(* IEC 61131-3 sources: SafePLC-Gen-Evaluation/Evaluation Results/eastman/run_05, 2 files *)

(* ---- io_declarations.st ---- *)
(* ==================================================  *)
(* PLC I/O Variable Declarations — CODESYS 3.5  *)
(* Generated by SafePLC-Gen Multimodal  *)
(* ==================================================  *)

VAR_GLOBAL
    (* --- Analog Inputs ---  *)
    FI_1_Raw                     AT %IW0       : INT := 0;    (* FI-1 — Flow indicator on feed/process line P-65  *)
    FI_2_Raw                     AT %IW2       : INT := 0;    (* FI-2 — Flow indicator on line P-54/P-52 area, f  *)
    FI_3_Raw                     AT %IW4       : INT := 0;    (* FI-3 — Flow indicator on line P-57 area, Column  *)
    TI_1_Raw                     AT %IW6       : INT := 0;    (* TI-1 — Temperature indicator, bottom-left area   *)
    TI_4_Raw                     AT %IW8       : INT := 0;    (* TI-4 — Temperature indicator on feed line to Co  *)
    TI_5_Raw                     AT %IW10      : INT := 0;    (* TI-5 — Temperature indicator on Column 2 (E-7),  *)
    TI_6_Raw                     AT %IW12      : INT := 0;    (* TI-6 — Temperature indicator on separator E-18   *)
    TI_7_Raw                     AT %IW14      : INT := 0;    (* TI-7 — Temperature indicator on Column 3 or ves  *)
    TI_8_Raw                     AT %IW16      : INT := 0;    (* TI-8 — Temperature indicator on Column 3, upper  *)
    (* --- Analog Outputs ---  *)
    V_3_Out                      AT %QW0       : INT := 0;    (* V-3 — Control valve on line P-28/P-73 from dec  *)
    V_4_Out                      AT %QW2       : INT := 0;    (* V-4 — Control valve on line P-74/P-12 feed to   *)
    V_5_Out                      AT %QW4       : INT := 0;    (* V-5 — Control valve on overhead/reflux line P-  *)
    V_7_Out                      AT %QW6       : INT := 0;    (* V-7 — Control valve on line P-19 from separato  *)
END_VAR

(* ---- generated_code.st ---- *)
(* Generated by SafePLC-Gen Multimodal — CODESYS 3.5 *)
(* IEC 61131-3 Structured Text *)
(* Date: 2026-04-25T12:43:58.560340 *)

PROGRAM DistillationControl

VAR
    FI_1_Raw                     AT %IW0       : INT := 0;
    FI_2_Raw                     AT %IW2       : INT := 0;
    FI_3_Raw                     AT %IW4       : INT := 0;
    TI_1_Raw                     AT %IW6       : INT := 0;
    TI_4_Raw                     AT %IW8       : INT := 0;
    TI_5_Raw                     AT %IW10      : INT := 0;
    TI_6_Raw                     AT %IW12      : INT := 0;
    TI_7_Raw                     AT %IW14      : INT := 0;
    TI_8_Raw                     AT %IW16      : INT := 0;
    V_3_Out                      AT %QW0       : INT := 0;
    V_4_Out                      AT %QW2       : INT := 0;
    V_5_Out                      AT %QW4       : INT := 0;
    V_7_Out                      AT %QW6       : INT := 0;
END_VAR

VAR
    FirstScan                    : BOOL := TRUE;

    FI_1_Scaled                  : REAL := 0.0;
    FI_2_Scaled                  : REAL := 0.0;
    FI_3_Scaled                  : REAL := 0.0;
    TI_1_Scaled                  : REAL := 0.0;
    TI_4_Scaled                  : REAL := 0.0;
    TI_5_Scaled                  : REAL := 0.0;
    TI_6_Scaled                  : REAL := 0.0;
    TI_7_Scaled                  : REAL := 0.0;
    TI_8_Scaled                  : REAL := 0.0;

    FI_1_HH_SP                   : REAL := 120.0;
    FI_1_H_SP                    : REAL := 100.0;
    FI_1_L_SP                    : REAL := 20.0;
    FI_1_LL_SP                   : REAL := 10.0;
    FI_1_Deadband                : REAL := 2.0;
    FI_1_HH                      : BOOL := FALSE;
    FI_1_H                       : BOOL := FALSE;
    FI_1_L                       : BOOL := FALSE;
    FI_1_LL                      : BOOL := FALSE;
    FI_1_HH_Latch                : SR := (S1 := FALSE, R := FALSE);
    FI_1_LL_Latch                : SR := (S1 := FALSE, R := FALSE);
    FI_1_HH_Ack                  : BOOL := FALSE;
    FI_1_LL_Ack                  : BOOL := FALSE;

    FI_2_HH_SP                   : REAL := 120.0;
    FI_2_H_SP                    : REAL := 100.0;
    FI_2_L_SP                    : REAL := 20.0;
    FI_2_LL_SP                   : REAL := 10.0;
    FI_2_Deadband                : REAL := 2.0;
    FI_2_HH                      : BOOL := FALSE;
    FI_2_H                       : BOOL := FALSE;
    FI_2_L                       : BOOL := FALSE;
    FI_2_LL                      : BOOL := FALSE;
    FI_2_HH_Latch                : SR := (S1 := FALSE, R := FALSE);
    FI_2_LL_Latch                : SR := (S1 := FALSE, R := FALSE);
    FI_2_HH_Ack                  : BOOL := FALSE;
    FI_2_LL_Ack                  : BOOL := FALSE;

    FI_3_HH_SP                   : REAL := 120.0;
    FI_3_H_SP                    : REAL := 100.0;
    FI_3_L_SP                    : REAL := 20.0;
    FI_3_LL_SP                   : REAL := 10.0;
    FI_3_Deadband                : REAL := 2.0;
    FI_3_HH                      : BOOL := FALSE;
    FI_3_H                       : BOOL := FALSE;
    FI_3_L                       : BOOL := FALSE;
    FI_3_LL                      : BOOL := FALSE;
    FI_3_HH_Latch                : SR := (S1 := FALSE, R := FALSE);
    FI_3_LL_Latch                : SR := (S1 := FALSE, R := FALSE);
    FI_3_HH_Ack                  : BOOL := FALSE;
    FI_3_LL_Ack                  : BOOL := FALSE;

    TI_1_HH_SP                   : REAL := 120.0;
    TI_1_H_SP                    : REAL := 110.0;
    TI_1_L_SP                    : REAL := 40.0;
    TI_1_LL_SP                   : REAL := 30.0;
    TI_1_Deadband                : REAL := 1.0;
    TI_1_HH                      : BOOL := FALSE;
    TI_1_H                       : BOOL := FALSE;
    TI_1_L                       : BOOL := FALSE;
    TI_1_LL                      : BOOL := FALSE;
    TI_1_HH_Latch                : SR := (S1 := FALSE, R := FALSE);
    TI_1_LL_Latch                : SR := (S1 := FALSE, R := FALSE);
    TI_1_HH_Ack                  : BOOL := FALSE;
    TI_1_LL_Ack                  : BOOL := FALSE;

    TI_4_HH_SP                   : REAL := 120.0;
    TI_4_H_SP                    : REAL := 110.0;
    TI_4_L_SP                    : REAL := 40.0;
    TI_4_LL_SP                   : REAL := 30.0;
    TI_4_Deadband                : REAL := 1.0;
    TI_4_HH                      : BOOL := FALSE;
    TI_4_H                       : BOOL := FALSE;
    TI_4_L                       : BOOL := FALSE;
    TI_4_LL                      : BOOL := FALSE;
    TI_4_HH_Latch                : SR := (S1 := FALSE, R := FALSE);
    TI_4_LL_Latch                : SR := (S1 := FALSE, R := FALSE);
    TI_4_HH_Ack                  : BOOL := FALSE;
    TI_4_LL_Ack                  : BOOL := FALSE;

    TI_5_HH_SP                   : REAL := 120.0;
    TI_5_H_SP                    : REAL := 110.0;
    TI_5_L_SP                    : REAL := 40.0;
    TI_5_LL_SP                   : REAL := 30.0;
    TI_5_Deadband                : REAL := 1.0;
    TI_5_HH                      : BOOL := FALSE;
    TI_5_H                       : BOOL := FALSE;
    TI_5_L                       : BOOL := FALSE;
    TI_5_LL                      : BOOL := FALSE;
    TI_5_HH_Latch                : SR := (S1 := FALSE, R := FALSE);
    TI_5_LL_Latch                : SR := (S1 := FALSE, R := FALSE);
    TI_5_HH_Ack                  : BOOL := FALSE;
    TI_5_LL_Ack                  : BOOL := FALSE;

    TI_6_HH_SP                   : REAL := 120.0;
    TI_6_H_SP                    : REAL := 110.0;
    TI_6_L_SP                    : REAL := 40.0;
    TI_6_LL_SP                   : REAL := 30.0;
    TI_6_Deadband                : REAL := 1.0;
    TI_6_HH                      : BOOL := FALSE;
    TI_6_H                       : BOOL := FALSE;
    TI_6_L                       : BOOL := FALSE;
    TI_6_LL                      : BOOL := FALSE;
    TI_6_HH_Latch                : SR := (S1 := FALSE, R := FALSE);
    TI_6_LL_Latch                : SR := (S1 := FALSE, R := FALSE);
    TI_6_HH_Ack                  : BOOL := FALSE;
    TI_6_LL_Ack                  : BOOL := FALSE;

    TI_7_HH_SP                   : REAL := 120.0;
    TI_7_H_SP                    : REAL := 110.0;
    TI_7_L_SP                    : REAL := 40.0;
    TI_7_LL_SP                   : REAL := 30.0;
    TI_7_Deadband                : REAL := 1.0;
    TI_7_HH                      : BOOL := FALSE;
    TI_7_H                       : BOOL := FALSE;
    TI_7_L                       : BOOL := FALSE;
    TI_7_LL                      : BOOL := FALSE;
    TI_7_HH_Latch                : SR := (S1 := FALSE, R := FALSE);
    TI_7_LL_Latch                : SR := (S1 := FALSE, R := FALSE);
    TI_7_HH_Ack                  : BOOL := FALSE;
    TI_7_LL_Ack                  : BOOL := FALSE;

    TI_8_HH_SP                   : REAL := 120.0;
    TI_8_H_SP                    : REAL := 110.0;
    TI_8_L_SP                    : REAL := 40.0;
    TI_8_LL_SP                   : REAL := 30.0;
    TI_8_Deadband                : REAL := 1.0;
    TI_8_HH                      : BOOL := FALSE;
    TI_8_H                       : BOOL := FALSE;
    TI_8_L                       : BOOL := FALSE;
    TI_8_LL                      : BOOL := FALSE;
    TI_8_HH_Latch                : SR := (S1 := FALSE, R := FALSE);
    TI_8_LL_Latch                : SR := (S1 := FALSE, R := FALSE);
    TI_8_HH_Ack                  : BOOL := FALSE;
    TI_8_LL_Ack                  : BOOL := FALSE;

    FC1_SP                       : REAL := 50.0;
    FC1_Kp                       : REAL := 1.2;
    FC1_Ki                       : REAL := 0.05;
    FC1_Error                    : REAL := 0.0;
    FC1_Integral                 : REAL := 0.0;
    FC1_Output                   : REAL := 0.0;

    FC2_SP                       : REAL := 50.0;
    FC2_Kp                       : REAL := 1.2;
    FC2_Ki                       : REAL := 0.05;
    FC2_Error                    : REAL := 0.0;
    FC2_Integral                 : REAL := 0.0;
    FC2_Output                   : REAL := 0.0;

    FC3_SP                       : REAL := 50.0;
    FC3_Kp                       : REAL := 1.2;
    FC3_Ki                       : REAL := 0.05;
    FC3_Error                    : REAL := 0.0;
    FC3_Integral                 : REAL := 0.0;
    FC3_Output                   : REAL := 0.0;

    TC1_SP                       : REAL := 80.0;
    TC1_Kp                       : REAL := 1.0;
    TC1_Ki                       : REAL := 0.03;
    TC1_Error                    : REAL := 0.0;
    TC1_Integral                 : REAL := 0.0;
    TC1_Output                   : REAL := 0.0;

    System_Alarm                 : BOOL := FALSE;
END_VAR

IF FirstScan THEN
    V_3_Out          := 6554;
    V_4_Out          := 6554;
    V_5_Out          := 6554;
    V_7_Out          := 6554;
    FC1_Integral     := 0.0;
    FC2_Integral     := 0.0;
    FC3_Integral     := 0.0;
    TC1_Integral     := 0.0;
    FI_1_HH_Latch(S1 := FALSE, R := FALSE);
    FI_1_LL_Latch(S1 := FALSE, R := FALSE);
    FI_2_HH_Latch(S1 := FALSE, R := FALSE);
    FI_2_LL_Latch(S1 := FALSE, R := FALSE);
    FI_3_HH_Latch(S1 := FALSE, R := FALSE);
    FI_3_LL_Latch(S1 := FALSE, R := FALSE);
    TI_1_HH_Latch(S1 := FALSE, R := FALSE);
    TI_1_LL_Latch(S1 := FALSE, R := FALSE);
    TI_4_HH_Latch(S1 := FALSE, R := FALSE);
    TI_4_LL_Latch(S1 := FALSE, R := FALSE);
    TI_5_HH_Latch(S1 := FALSE, R := FALSE);
    TI_5_LL_Latch(S1 := FALSE, R := FALSE);
    TI_6_HH_Latch(S1 := FALSE, R := FALSE);
    TI_6_LL_Latch(S1 := FALSE, R := FALSE);
    TI_7_HH_Latch(S1 := FALSE, R := FALSE);
    TI_7_LL_Latch(S1 := FALSE, R := FALSE);
    TI_8_HH_Latch(S1 := FALSE, R := FALSE);
    TI_8_LL_Latch(S1 := FALSE, R := FALSE);
    FirstScan        := FALSE;
    RETURN;
END_IF;

FI_1_Scaled := ((INT_TO_REAL(FI_1_Raw) - 6554.0) / (32767.0 - 6554.0)) * 150.0;
FI_2_Scaled := ((INT_TO_REAL(FI_2_Raw) - 6554.0) / (32767.0 - 6554.0)) * 150.0;
FI_3_Scaled := ((INT_TO_REAL(FI_3_Raw) - 6554.0) / (32767.0 - 6554.0)) * 150.0;
TI_1_Scaled := ((INT_TO_REAL(TI_1_Raw) - 6554.0) / (32767.0 - 6554.0)) * 150.0;
TI_4_Scaled := ((INT_TO_REAL(TI_4_Raw) - 6554.0) / (32767.0 - 6554.0)) * 150.0;
TI_5_Scaled := ((INT_TO_REAL(TI_5_Raw) - 6554.0) / (32767.0 - 6554.0)) * 150.0;
TI_6_Scaled := ((INT_TO_REAL(TI_6_Raw) - 6554.0) / (32767.0 - 6554.0)) * 150.0;
TI_7_Scaled := ((INT_TO_REAL(TI_7_Raw) - 6554.0) / (32767.0 - 6554.0)) * 150.0;
TI_8_Scaled := ((INT_TO_REAL(TI_8_Raw) - 6554.0) / (32767.0 - 6554.0)) * 150.0;

IF FI_1_Scaled >= FI_1_HH_SP THEN
    FI_1_HH_Latch.S1 := TRUE;
ELSIF FI_1_Scaled <= (FI_1_HH_SP - FI_1_Deadband) THEN
    FI_1_HH_Latch.S1 := FALSE;
END_IF;
FI_1_HH_Latch.R := FI_1_HH_Ack AND (FI_1_Scaled < FI_1_HH_SP);
FI_1_HH_Latch(S1 := FI_1_HH_Latch.S1, R := FI_1_HH_Latch.R);
FI_1_HH := FI_1_HH_Latch.Q1;

IF FI_1_Scaled >= FI_1_H_SP THEN
    FI_1_H := TRUE;
ELSIF FI_1_Scaled < (FI_1_H_SP - FI_1_Deadband) THEN
    FI_1_H := FALSE;
END_IF;

IF FI_1_Scaled <= FI_1_LL_SP THEN
    FI_1_LL_Latch.S1 := TRUE;
ELSIF FI_1_Scaled >= (FI_1_LL_SP + FI_1_Deadband) THEN
    FI_1_LL_Latch.S1 := FALSE;
END_IF;
FI_1_LL_Latch.R := FI_1_LL_Ack AND (FI_1_Scaled > FI_1_LL_SP);
FI_1_LL_Latch(S1 := FI_1_LL_Latch.S1, R := FI_1_LL_Latch.R);
FI_1_LL := FI_1_LL_Latch.Q1;

IF FI_1_Scaled <= FI_1_L_SP THEN
    FI_1_L := TRUE;
ELSIF FI_1_Scaled > (FI_1_L_SP + FI_1_Deadband) THEN
    FI_1_L := FALSE;
END_IF;

IF FI_2_Scaled >= FI_2_HH_SP THEN
    FI_2_HH_Latch.S1 := TRUE;
ELSIF FI_2_Scaled <= (FI_2_HH_SP - FI_2_Deadband) THEN
    FI_2_HH_Latch.S1 := FALSE;
END_IF;
FI_2_HH_Latch.R := FI_2_HH_Ack AND (FI_2_Scaled < FI_2_HH_SP);
FI_2_HH_Latch(S1 := FI_2_HH_Latch.S1, R := FI_2_HH_Latch.R);
FI_2_HH := FI_2_HH_Latch.Q1;

IF FI_2_Scaled >= FI_2_H_SP THEN
    FI_2_H := TRUE;
ELSIF FI_2_Scaled < (FI_2_H_SP - FI_2_Deadband) THEN
    FI_2_H := FALSE;
END_IF;

IF FI_2_Scaled <= FI_2_LL_SP THEN
    FI_2_LL_Latch.S1 := TRUE;
ELSIF FI_2_Scaled >= (FI_2_LL_SP + FI_2_Deadband) THEN
    FI_2_LL_Latch.S1 := FALSE;
END_IF;
FI_2_LL_Latch.R := FI_2_LL_Ack AND (FI_2_Scaled > FI_2_LL_SP);
FI_2_LL_Latch(S1 := FI_2_LL_Latch.S1, R := FI_2_LL_Latch.R);
FI_2_LL := FI_2_LL_Latch.Q1;

IF FI_2_Scaled <= FI_2_L_SP THEN
    FI_2_L := TRUE;
ELSIF FI_2_Scaled > (FI_2_L_SP + FI_2_Deadband) THEN
    FI_2_L := FALSE;
END_IF;

IF FI_3_Scaled >= FI_3_HH_SP THEN
    FI_3_HH_Latch.S1 := TRUE;
ELSIF FI_3_Scaled <= (FI_3_HH_SP - FI_3_Deadband) THEN
    FI_3_HH_Latch.S1 := FALSE;
END_IF;
FI_3_HH_Latch.R := FI_3_HH_Ack AND (FI_3_Scaled < FI_3_HH_SP);
FI_3_HH_Latch(S1 := FI_3_HH_Latch.S1, R := FI_3_HH_Latch.R);
FI_3_HH := FI_3_HH_Latch.Q1;

IF FI_3_Scaled >= FI_3_H_SP THEN
    FI_3_H := TRUE;
ELSIF FI_3_Scaled < (FI_3_H_SP - FI_3_Deadband) THEN
    FI_3_H := FALSE;
END_IF;

IF FI_3_Scaled <= FI_3_LL_SP THEN
    FI_3_LL_Latch.S1 := TRUE;
ELSIF FI_3_Scaled >= (FI_3_LL_SP + FI_3_Deadband) THEN
    FI_3_LL_Latch.S1 := FALSE;
END_IF;
FI_3_LL_Latch.R := FI_3_LL_Ack AND (FI_3_Scaled > FI_3_LL_SP);
FI_3_LL_Latch(S1 := FI_3_LL_Latch.S1, R := FI_3_LL_Latch.R);
FI_3_LL := FI_3_LL_Latch.Q1;

IF FI_3_Scaled <= FI_3_L_SP THEN
    FI_3_L := TRUE;
ELSIF FI_3_Scaled > (FI_3_L_SP + FI_3_Deadband) THEN
    FI_3_L := FALSE;
END_IF;

IF TI_1_Scaled >= TI_1_HH_SP THEN
    TI_1_HH_Latch.S1 := TRUE;
ELSIF TI_1_Scaled <= (TI_1_HH_SP - TI_1_Deadband) THEN
    TI_1_HH_Latch.S1 := FALSE;
END_IF;
TI_1_HH_Latch.R := TI_1_HH_Ack AND (TI_1_Scaled < TI_1_HH_SP);
TI_1_HH_Latch(S1 := TI_1_HH_Latch.S1, R := TI_1_HH_Latch.R);
TI_1_HH := TI_1_HH_Latch.Q1;

IF TI_1_Scaled >= TI_1_H_SP THEN
    TI_1_H := TRUE;
ELSIF TI_1_Scaled < (TI_1_H_SP - TI_1_Deadband) THEN
    TI_1_H := FALSE;
END_IF;

IF TI_1_Scaled <= TI_1_LL_SP THEN
    TI_1_LL_Latch.S1 := TRUE;
ELSIF TI_1_Scaled >= (TI_1_LL_SP + TI_1_Deadband) THEN
    TI_1_LL_Latch.S1 := FALSE;
END_IF;
TI_1_LL_Latch.R := TI_1_LL_Ack AND (TI_1_Scaled > TI_1_LL_SP);
TI_1_LL_Latch(S1 := TI_1_LL_Latch.S1, R := TI_1_LL_Latch.R);
TI_1_LL := TI_1_LL_Latch.Q1;

IF TI_1_Scaled <= TI_1_L_SP THEN
    TI_1_L := TRUE;
ELSIF TI_1_Scaled > (TI_1_L_SP + TI_1_Deadband) THEN
    TI_1_L := FALSE;
END_IF;

IF TI_4_Scaled >= TI_4_HH_SP THEN
    TI_4_HH_Latch.S1 := TRUE;
ELSIF TI_4_Scaled <= (TI_4_HH_SP - TI_4_Deadband) THEN
    TI_4_HH_Latch.S1 := FALSE;
END_IF;
TI_4_HH_Latch.R := TI_4_HH_Ack AND (TI_4_Scaled < TI_4_HH_SP);
TI_4_HH_Latch(S1 := TI_4_HH_Latch.S1, R := TI_4_HH_Latch.R);
TI_4_HH := TI_4_HH_Latch.Q1;

IF TI_4_Scaled >= TI_4_H_SP THEN
    TI_4_H := TRUE;
ELSIF TI_4_Scaled < (TI_4_H_SP - TI_4_Deadband) THEN
    TI_4_H := FALSE;
END_IF;

IF TI_4_Scaled <= TI_4_LL_SP THEN
    TI_4_LL_Latch.S1 := TRUE;
ELSIF TI_4_Scaled >= (TI_4_LL_SP + TI_4_Deadband) THEN
    TI_4_LL_Latch.S1 := FALSE;
END_IF;
TI_4_LL_Latch.R := TI_4_LL_Ack AND (TI_4_Scaled > TI_4_LL_SP);
TI_4_LL_Latch(S1 := TI_4_LL_Latch.S1, R := TI_4_LL_Latch.R);
TI_4_LL := TI_4_LL_Latch.Q1;

IF TI_4_Scaled <= TI_4_L_SP THEN
    TI_4_L := TRUE;
ELSIF TI_4_Scaled > (TI_4_L_SP + TI_4_Deadband) THEN
    TI_4_L := FALSE;
END_IF;

IF TI_5_Scaled >= TI_5_HH_SP THEN
    TI_5_HH_Latch.S1 := TRUE;
ELSIF TI_5_Scaled <= (TI_5_HH_SP - TI_5_Deadband) THEN
    TI_5_HH_Latch.S1 := FALSE;
END_IF;
TI_5_HH_Latch.R := TI_5_HH_Ack AND (TI_5_Scaled < TI_5_HH_SP);
TI_5_HH_Latch(S1 := TI_5_HH_Latch.S1, R := TI_5_HH_Latch.R);
TI_5_HH := TI_5_HH_Latch.Q1;

IF TI_5_Scaled >= TI_5_H_SP THEN
    TI_5_H := TRUE;
ELSIF TI_5_Scaled < (TI_5_H_SP - TI_5_Deadband) THEN
    TI_5_H := FALSE;
END_IF;

IF TI_5_Scaled <= TI_5_LL_SP THEN
    TI_5_LL_Latch.S1 := TRUE;
ELSIF TI_5_Scaled >= (TI_5_LL_SP + TI_5_Deadband) THEN
    TI_5_LL_Latch.S1 := FALSE;
END_IF;
TI_5_LL_Latch.R := TI_5_LL_Ack AND (TI_5_Scaled > TI_5_LL_SP);
TI_5_LL_Latch(S1 := TI_5_LL_Latch.S1, R := TI_5_LL_Latch.R);
TI_5_LL := TI_5_LL_Latch.Q1;

IF TI_5_Scaled <= TI_5_L_SP THEN
    TI_5_L := TRUE;
ELSIF TI_5_Scaled > (TI_5_L_SP + TI_5_Deadband) THEN
    TI_5_L := FALSE;
END_IF;

IF TI_6_Scaled >= TI_6_HH_SP THEN
    TI_6_HH_Latch.S1 := TRUE;
ELSIF TI_6_Scaled <= (TI_6_HH_SP - TI_6_Deadband) THEN
    TI_6_HH_Latch.S1 := FALSE;
END_IF;
TI_6_HH_Latch.R := TI_6_HH_Ack AND (TI_6_Scaled < TI_6_HH_SP);
TI_6_HH_Latch(S1 := TI_6_HH_Latch.S1, R := TI_6_HH_Latch.R);
TI_6_HH := TI_6_HH_Latch.Q1;

IF TI_6_Scaled >= TI_6_H_SP THEN
    TI_6_H := TRUE;
ELSIF TI_6_Scaled < (TI_6_H_SP - TI_6_Deadband) THEN
    TI_6_H := FALSE;
END_IF;

IF TI_6_Scaled <= TI_6_LL_SP THEN
    TI_6_LL_Latch.S1 := TRUE;
ELSIF TI_6_Scaled >= (TI_6_LL_SP + TI_6_Deadband) THEN
    TI_6_LL_Latch.S1 := FALSE;
END_IF;
TI_6_LL_Latch.R := TI_6_LL_Ack AND (TI_6_Scaled > TI_6_LL_SP);
TI_6_LL_Latch(S1 := TI_6_LL_Latch.S1, R := TI_6_LL_Latch.R);
TI_6_LL := TI_6_LL_Latch.Q1;

IF TI_6_Scaled <= TI_6_L_SP THEN
    TI_6_L := TRUE;
ELSIF TI_6_Scaled > (TI_6_L_SP + TI_6_Deadband) THEN
    TI_6_L := FALSE;
END_IF;

IF TI_7_Scaled >= TI_7_HH_SP THEN
    TI_7_HH_Latch.S1 := TRUE;
ELSIF TI_7_Scaled <= (TI_7_HH_SP - TI_7_Deadband) THEN
    TI_7_HH_Latch.S1 := FALSE;
END_IF;
TI_7_HH_Latch.R := TI_7_HH_Ack AND (TI_7_Scaled < TI_7_HH_SP);
TI_7_HH_Latch(S1 := TI_7_HH_Latch.S1, R := TI_7_HH_Latch.R);
TI_7_HH := TI_7_HH_Latch.Q1;

IF TI_7_Scaled >= TI_7_H_SP THEN
    TI_7_H := TRUE;
ELSIF TI_7_Scaled < (TI_7_H_SP - TI_7_Deadband) THEN
    TI_7_H := FALSE;
END_IF;

IF TI_7_Scaled <= TI_7_LL_SP THEN
    TI_7_LL_Latch.S1 := TRUE;
ELSIF TI_7_Scaled >= (TI_7_LL_SP + TI_7_Deadband) THEN
    TI_7_LL_Latch.S1 := FALSE;
END_IF;
TI_7_LL_Latch.R := TI_7_LL_Ack AND (TI_7_Scaled > TI_7_LL_SP);
TI_7_LL_Latch(S1 := TI_7_LL_Latch.S1, R := TI_7_LL_Latch.R);
TI_7_LL := TI_7_LL_Latch.Q1;

IF TI_7_Scaled <= TI_7_L_SP THEN
    TI_7_L := TRUE;
ELSIF TI_7_Scaled > (TI_7_L_SP + TI_7_Deadband) THEN
    TI_7_L := FALSE;
END_IF;

IF TI_8_Scaled >= TI_8_HH_SP THEN
    TI_8_HH_Latch.S1 := TRUE;
ELSIF TI_8_Scaled <= (TI_8_HH_SP - TI_8_Deadband) THEN
    TI_8_HH_Latch.S1 := FALSE;
END_IF;
TI_8_HH_Latch.R := TI_8_HH_Ack AND (TI_8_Scaled < TI_8_HH_SP);
TI_8_HH_Latch(S1 := TI_8_HH_Latch.S1, R := TI_8_HH_Latch.R);
TI_8_HH := TI_8_HH_Latch.Q1;

IF TI_8_Scaled >= TI_8_H_SP THEN
    TI_8_H := TRUE;
ELSIF TI_8_Scaled < (TI_8_H_SP - TI_8_Deadband) THEN
    TI_8_H := FALSE;
END_IF;

IF TI_8_Scaled <= TI_8_LL_SP THEN
    TI_8_LL_Latch.S1 := TRUE;
ELSIF TI_8_Scaled >= (TI_8_LL_SP + TI_8_Deadband) THEN
    TI_8_LL_Latch.S1 := FALSE;
END_IF;
TI_8_LL_Latch.R := TI_8_LL_Ack AND (TI_8_Scaled > TI_8_LL_SP);
TI_8_LL_Latch(S1 := TI_8_LL_Latch.S1, R := TI_8_LL_Latch.R);
TI_8_LL := TI_8_LL_Latch.Q1;

IF TI_8_Scaled <= TI_8_L_SP THEN
    TI_8_L := TRUE;
ELSIF TI_8_Scaled > (TI_8_L_SP + TI_8_Deadband) THEN
    TI_8_L := FALSE;
END_IF;

FC1_Error    := FC1_SP - FI_1_Scaled;
FC1_Integral := FC1_Integral + (FC1_Ki * FC1_Error);
IF FC1_Integral > 100.0 THEN
    FC1_Integral := 100.0;
ELSIF FC1_Integral < 0.0 THEN
    FC1_Integral := 0.0;
END_IF;
FC1_Output := (FC1_Kp * FC1_Error) + FC1_Integral;
IF FC1_Output > 100.0 THEN
    FC1_Output := 100.0;
ELSIF FC1_Output < 0.0 THEN
    FC1_Output := 0.0;
END_IF;
V_3_Out := REAL_TO_INT(6554.0 + (FC1_Output / 100.0) * (32767.0 - 6554.0));

FC2_Error    := FC2_SP - FI_2_Scaled;
FC2_Integral := FC2_Integral + (FC2_Ki * FC2_Error);
IF FC2_Integral > 100.0 THEN
    FC2_Integral := 100.0;
ELSIF FC2_Integral < 0.0 THEN
    FC2_Integral := 0.0;
END_IF;
FC2_Output := (FC2_Kp * FC2_Error) + FC2_Integral;
IF FC2_Output > 100.0 THEN
    FC2_Output := 100.0;
ELSIF FC2_Output < 0.0 THEN
    FC2_Output := 0.0;
END_IF;
V_4_Out := REAL_TO_INT(6554.0 + (FC2_Output / 100.0) * (32767.0 - 6554.0));

FC3_Error    := FC3_SP - FI_3_Scaled;
FC3_Integral := FC3_Integral + (FC3_Ki * FC3_Error);
IF FC3_Integral > 100.0 THEN
    FC3_Integral := 100.0;
ELSIF FC3_Integral < 0.0 THEN
    FC3_Integral := 0.0;
END_IF;
FC3_Output := (FC3_Kp * FC3_Error) + FC3_Integral;
IF FC3_Output > 100.0 THEN
    FC3_Output := 100.0;
ELSIF FC3_Output < 0.0 THEN
    FC3_Output := 0.0;
END_IF;
V_5_Out := REAL_TO_INT(6554.0 + (FC3_Output / 100.0) * (32767.0 - 6554.0));

TC1_Error    := TC1_SP - TI_4_Scaled;
TC1_Integral := TC1_Integral + (TC1_Ki * TC1_Error);
IF TC1_Integral > 100.0 THEN
    TC1_Integral := 100.0;
ELSIF TC1_Integral < 0.0 THEN
    TC1_Integral := 0.0;
END_IF;
TC1_Output := (TC1_Kp * TC1_Error) + TC1_Integral;
IF TC1_Output > 100.0 THEN
    TC1_Output := 100.0;
ELSIF TC1_Output < 0.0 THEN
    TC1_Output := 0.0;
END_IF;
V_7_Out := REAL_TO_INT(6554.0 + (TC1_Output / 100.0) * (32767.0 - 6554.0));

System_Alarm :=
    FI_1_HH_Latch.Q1 OR FI_1_LL_Latch.Q1 OR FI_1_H OR FI_1_L OR
    FI_2_HH_Latch.Q1 OR FI_2_LL_Latch.Q1 OR FI_2_H OR FI_2_L OR
    FI_3_HH_Latch.Q1 OR FI_3_LL_Latch.Q1 OR FI_3_H OR FI_3_L OR
    TI_1_HH_Latch.Q1 OR TI_1_LL_Latch.Q1 OR TI_1_H OR TI_1_L OR
    TI_4_HH_Latch.Q1 OR TI_4_LL_Latch.Q1 OR TI_4_H OR TI_4_L OR
    TI_5_HH_Latch.Q1 OR TI_5_LL_Latch.Q1 OR TI_5_H OR TI_5_L OR
    TI_6_HH_Latch.Q1 OR TI_6_LL_Latch.Q1 OR TI_6_H OR TI_6_L OR
    TI_7_HH_Latch.Q1 OR TI_7_LL_Latch.Q1 OR TI_7_H OR TI_7_L OR
    TI_8_HH_Latch.Q1 OR TI_8_LL_Latch.Q1 OR TI_8_H OR TI_8_L;

END_PROGRAM
